TYPE TelemetryStatuses :
STRUCT
	initializationStatus: InitializationStatus;
	healthStatus: HealthStatus;
	busyStatus: BusyStatus;
	operatingStatus: OperatingStatus;
END_STRUCT
END_TYPE

(* stored: Version 1.1.0.1, ProductVersion 3.1.4019.2
   DUT TelemetryStatuses: Id {03215b41-7f1d-4f92-8f4f-e189292a5b0d} *)
